FUNCTION FC_SQL_InsertCommands_Encoder : STRING(255)
VAR_INPUT
    iSensorValue: LREAL;
    iSampleNr: INT;
	iMeasurementNr: INT;
END_VAR

FC_SQL_InsertCommands_Encoder := 'INSERT INTO [db_accessadmin].[Encoder] (SensorValue, SampleNr, Time, MeasurementNr) VALUES (';
FC_SQL_InsertCommands_Encoder := CONCAT(FC_SQL_InsertCommands_Encoder, LREAL_TO_STRING(iSensorValue));
FC_SQL_InsertCommands_Encoder := CONCAT(FC_SQL_InsertCommands_Encoder, ', ');
FC_SQL_InsertCommands_Encoder := CONCAT(FC_SQL_InsertCommands_Encoder, INT_TO_STRING(iSampleNr));
FC_SQL_InsertCommands_Encoder := CONCAT(FC_SQL_InsertCommands_Encoder, ', GETDATE() ');
FC_SQL_InsertCommands_Encoder := CONCAT(FC_SQL_InsertCommands_Encoder, ', ');
FC_SQL_InsertCommands_Encoder := CONCAT(FC_SQL_InsertCommands_Encoder, INT_TO_STRING(iMeasurementNr));
FC_SQL_InsertCommands_Encoder := CONCAT(FC_SQL_InsertCommands_Encoder, ');');

END_FUNCTION

(* stored: Version 1.1.0.1
   POU FC_SQL_InsertCommands_Encoder: Id {4243be30-0310-4c85-bbee-74be1aa1fdb2}, SpecialFunc None *)
